FUNCTION_BLOCK _ETcVn2dCodeSearchStrategy_TestSuite EXTENDS TcUnit.FB_TestSuite
VAR
END_VAR

TestAddress();
TestClearReference();
TestClone();
TestTypeNameReturnsExpected();
TestIdentifierReturnsExpected();
TestMakeReferenceToFollowsReference();
TestMakeReferenceToUpdatesReference();
TestSize();
TestValueReturnsExpectedAfterInit();
TestValueReturnsExpectedAfterChange();
TestSerializeTypeWith();
TestSerializeWith();
TestTryDeserializeFrom();
TestTryMakeReferenceToFollowsReference();
TestTryMakeReferenceToUpdatesReference();

METHOD PUBLIC TestAddress
VAR
    _type : _ETcVn2dCodeSearchStrategy(ETcVn2dCodeSearchStrategy.TCVN_CSS_DEFAULT);
    notExpected : PVOID := 0;
    actual : PVOID;
END_VAR
TEST('TestAddress');

actual := _type.Address;

AssertFalse(
    Condition := (notExpected = actual),
    Message := 'Type did not return a valid address.'
);

TEST_FINISHED();
END_METHOD

METHOD PUBLIC TestClearReference
VAR
    _type : _ETcVn2dCodeSearchStrategy(ETcVn2dCodeSearchStrategy.TCVN_CSS_DEFAULT);
	target : ETcVn2dCodeSearchStrategy := ETcVn2dCodeSearchStrategy.TCVN_CSS_DEFAULT;
    expected : ETcVn2dCodeSearchStrategy := ETcVn2dCodeSearchStrategy.TCVN_CSS_DEFAULT;
    actual : ETcVn2dCodeSearchStrategy;
END_VAR
TEST('TestClearReference');

_type.MakeReferenceTo(target);
_type.ClearReference();
target := ETcVn2dCodeSearchStrategy.TCVN_CSS_FIRST_FLIPPED;

actual := _type.Value;

AssertEquals(
    Expected := expected,
    Actual := actual,
    Message := 'Value continued to follow target.'
);

TEST_FINISHED();
END_METHOD

METHOD PUBLIC TestClone
VAR
    _type : _ETcVn2dCodeSearchStrategy(ETcVn2dCodeSearchStrategy.TCVN_CSS_DEFAULT);
	clone : I_Datatype;
	isValidClone : BOOL;
	compareResult : DINT;
END_VAR
TEST('TestClone');

clone := _type.Clone();

isValidClone := clone <> 0;

IF isValidClone THEN
	compareResult := memcmp(_type.Address, clone.Address, clone.Size);
END_IF

AssertTrue(
	Condition := isValidClone,
	Message := 'Clone did not produce a clone'
);

AssertEquals_DINT(
	Expected := 0,
    Actual := compareResult,
    Message := 'Clone did not return a valid clone.'
);

clone.Dispose();

TEST_FINISHED();
END_METHOD

METHOD PUBLIC TestIdentifierReturnsExpected
VAR
    _type : _ETcVn2dCodeSearchStrategy(ETcVn2dCodeSearchStrategy.TCVN_CSS_DEFAULT);
    expected : STRING := 'ETcVn2dCodeSearchStrategy';
    actual : STRING;
END_VAR
TEST('TestIdentifierReturnsExpected');

actual := _type.Identifier;

AssertEquals_STRING(
    Expected := expected,
    Actual := actual,
    Message := 'Type did not return correct iec type.'
);

TEST_FINISHED();
END_METHOD

METHOD PUBLIC TestMakeReferenceToFollowsReference
VAR
    _type : _ETcVn2dCodeSearchStrategy(ETcVn2dCodeSearchStrategy.TCVN_CSS_DEFAULT);
	target : ETcVn2dCodeSearchStrategy := ETcVn2dCodeSearchStrategy.TCVN_CSS_DEFAULT;
    expected : ETcVn2dCodeSearchStrategy := ETcVn2dCodeSearchStrategy.TCVN_CSS_FIRST_FLIPPED;
    actual : ETcVn2dCodeSearchStrategy;
END_VAR
TEST('TestMakeReferenceToFollowsReference');

_type.MakeReferenceTo(target);
target := ETcVn2dCodeSearchStrategy.TCVN_CSS_FIRST_FLIPPED;

actual := _type.Value;

AssertEquals(
    Expected := expected,
    Actual := actual,
    Message := 'Value did not follow target change.'
);

TEST_FINISHED();
END_METHOD

METHOD PUBLIC TestMakeReferenceToUpdatesReference
VAR
    _type : _ETcVn2dCodeSearchStrategy(ETcVn2dCodeSearchStrategy.TCVN_CSS_DEFAULT);
	target : ETcVn2dCodeSearchStrategy := ETcVn2dCodeSearchStrategy.TCVN_CSS_DEFAULT;
    expected : ETcVn2dCodeSearchStrategy := ETcVn2dCodeSearchStrategy.TCVN_CSS_FIRST_FLIPPED;
    actual : ETcVn2dCodeSearchStrategy;
END_VAR
TEST('TestMakeReferenceToUpdatesReference');

_type.MakeReferenceTo(target);
_type.Value := ETcVn2dCodeSearchStrategy.TCVN_CSS_FIRST_FLIPPED;

actual := target;

AssertEquals(
    Expected := expected,
    Actual := actual,
    Message := 'Value did not update target.'
);

TEST_FINISHED();
END_METHOD

METHOD PUBLIC TestSerializeTypeWith
VAR
    _type : _ETcVn2dCodeSearchStrategy(ETcVn2dCodeSearchStrategy.TCVN_CSS_DEFAULT);
    serializer : JsonSerializer;
    expected : STRING(500) := '{"typeName":"ENUM","identifier":"ETcVn2dCodeSearchStrategy","enumerations":["TCVN_CSS_DEFAULT","TCVN_CSS_FIRST_FLIPPED","TCVN_CSS_FIRST_INVERTED","TCVN_CSS_FIRST_NOT_FLIPPED","TCVN_CSS_FIRST_NOT_INVERTED","TCVN_CSS_ONLY_FLIPPED","TCVN_CSS_ONLY_INVERTED","TCVN_CSS_ONLY_NOT_FLIPPED","TCVN_CSS_ONLY_NOT_INVERTED"],"baseType":{"typeName":"UDINT","minValue":0,"maxValue":4294967295,"isSigned":false,"isFloat":false}}';
    actual : STRING(500);
END_VAR
TEST('TestSerializeTypeWith');

serializer.Reset();
_type.SerializeTypeWith(serializer);
serializer.TryGetSerializedData(ADR(actual), SIZEOF(actual));

AssertEquals_STRING(
    Expected := expected,
    Actual := actual,
    Message := 'Serialization of type did not return correct string.'
);

TEST_FINISHED();
END_METHOD

METHOD PUBLIC TestSerializeWith
VAR
    _type : _ETcVn2dCodeSearchStrategy(ETcVn2dCodeSearchStrategy.TCVN_CSS_DEFAULT);
    serializer : JsonSerializer;
    expected : STRING := '"TCVN_CSS_DEFAULT"';
    actual : STRING(500);
END_VAR
TEST('TestSerializeWith');

serializer.Reset();
_type.SerializeWith(serializer);
serializer.TryGetSerializedData(ADR(actual), SIZEOF(actual));

AssertEquals_STRING(
    Expected := expected,
    Actual := actual,
    Message := 'Serialization of type data did not return correct string.'
);

TEST_FINISHED();
END_METHOD

METHOD PUBLIC TestSize
VAR
    _type : _ETcVn2dCodeSearchStrategy(ETcVn2dCodeSearchStrategy.TCVN_CSS_DEFAULT);
    expected : UDINT := SIZEOF(ETcVn2dCodeSearchStrategy);
    actual : UDINT;
END_VAR
TEST('TestSize');

actual := _type.Size;

AssertEquals_UDINT(
    Expected := Expected,
    Actual := actual,
    Message := 'Type did not return the correct size.'
);

TEST_FINISHED();
END_METHOD

METHOD PUBLIC TestTryDeserializeFrom
VAR
    deserializer : JsonDeserializer;
    feedback : DeserializerFeedback;
    json : STRING := '"TCVN_CSS_DEFAULT"';
    _type : _ETcVn2dCodeSearchStrategy(ETcVn2dCodeSearchStrategy.TCVN_CSS_DEFAULT);
    expected : ETcVn2dCodeSearchStrategy := ETcVn2dCodeSearchStrategy.TCVN_CSS_DEFAULT;
    actual : ETcVn2dCodeSearchStrategy;
 END_VAR
TEST('TestTryDeserializeFrom');

deserializer.Reset();
deserializer.TryLoad(json);
_type.TryDeserializeFrom(Deserializer, Feedback);

actual := _type.Value;

AssertEquals(
    Expected := expected,
    Actual := actual,
    Message := 'Type did not deserialize correctly.'
);

TEST_FINISHED();
END_METHOD

METHOD PUBLIC TestTryMakeReferenceToFollowsReference
VAR
    _type : _ETcVn2dCodeSearchStrategy(ETcVn2dCodeSearchStrategy.TCVN_CSS_DEFAULT);
	target : _ETcVn2dCodeSearchStrategy(ETcVn2dCodeSearchStrategy.TCVN_CSS_DEFAULT);
    expected : ETcVn2dCodeSearchStrategy := ETcVn2dCodeSearchStrategy.TCVN_CSS_FIRST_FLIPPED;
    actual : ETcVn2dCodeSearchStrategy;
END_VAR
TEST('TestTryMakeReferenceToFollowsReference');

_type.TryMakeReferenceTo(target);
target.Value := ETcVn2dCodeSearchStrategy.TCVN_CSS_FIRST_FLIPPED;

actual := _type.Value;

AssertEquals(
    Expected := expected,
    Actual := actual,
    Message := 'Value did not follow target change.'
);

TEST_FINISHED();
END_METHOD

METHOD PUBLIC TestTryMakeReferenceToUpdatesReference
VAR
    _type : _ETcVn2dCodeSearchStrategy(ETcVn2dCodeSearchStrategy.TCVN_CSS_DEFAULT);
	target : _ETcVn2dCodeSearchStrategy(ETcVn2dCodeSearchStrategy.TCVN_CSS_DEFAULT);
    expected : ETcVn2dCodeSearchStrategy := ETcVn2dCodeSearchStrategy.TCVN_CSS_FIRST_FLIPPED;
    actual : ETcVn2dCodeSearchStrategy;
END_VAR
TEST('TestTryMakeReferenceToUpdatesReference');

_type.TryMakeReferenceTo(target);
_type.Value := ETcVn2dCodeSearchStrategy.TCVN_CSS_FIRST_FLIPPED;

actual := target.Value;

AssertEquals(
    Expected := expected,
    Actual := actual,
    Message := 'Value did not update target.'
);

TEST_FINISHED();
END_METHOD

METHOD PUBLIC TestTypeNameReturnsExpected
VAR
    _type : _ETcVn2dCodeSearchStrategy(ETcVn2dCodeSearchStrategy.TCVN_CSS_DEFAULT);
    expected : STRING := 'ENUM';
    actual : STRING;
END_VAR
TEST('TestTypeNameReturnsExpected');

actual := _type.TypeName;

AssertEquals_STRING(
    Expected := expected,
    Actual := actual,
    Message := 'Type did not return correct iec type.'
);

TEST_FINISHED();
END_METHOD

METHOD PUBLIC TestValueReturnsExpectedAfterChange
VAR
    _type : _ETcVn2dCodeSearchStrategy(ETcVn2dCodeSearchStrategy.TCVN_CSS_DEFAULT);
    expected : ETcVn2dCodeSearchStrategy := ETcVn2dCodeSearchStrategy.TCVN_CSS_FIRST_FLIPPED;
    actual : ETcVn2dCodeSearchStrategy;
END_VAR
TEST('TestValueReturnsExpectedAfterChange');

_type.Value := ETcVn2dCodeSearchStrategy.TCVN_CSS_FIRST_FLIPPED;

actual := _type.Value;

AssertEquals(
    Expected := expected,
    Actual := actual,
    Message := 'Expected value not returned after change.'
);

TEST_FINISHED();
END_METHOD

METHOD PUBLIC TestValueReturnsExpectedAfterInit
VAR
    _type : _ETcVn2dCodeSearchStrategy(ETcVn2dCodeSearchStrategy.TCVN_CSS_DEFAULT);
    expected : ETcVn2dCodeSearchStrategy := ETcVn2dCodeSearchStrategy.TCVN_CSS_DEFAULT;
    actual : ETcVn2dCodeSearchStrategy;
END_VAR
TEST('TestValueReturnsExpectedAfterInit');

actual := _type.Value;

AssertEquals(
    Expected := expected,
    Actual := actual,
    Message := 'Expected value not returned after Init.'
);

TEST_FINISHED();
END_METHOD

END_FUNCTION_BLOCK

(* stored: Version 1.1.0.1, ProductVersion 3.1.4024.12
   POU _ETcVn2dCodeSearchStrategy_TestSuite: Id {6437228a-7660-4c0d-b535-65226c912a28}, SpecialFunc None
   Method TestAddress: Id {e5d5aed4-c00a-464d-ba41-6f769ea80945}
   Method TestClearReference: Id {ccb49ab5-497b-4333-82a4-81aca560be1f}
   Method TestClone: Id {f7783ad6-e504-428e-81a7-36fba43d27f4}
   Method TestIdentifierReturnsExpected: Id {a1efc315-531e-43d6-867b-93b1ce671e5d}
   Method TestMakeReferenceToFollowsReference: Id {0650108b-4755-438e-927b-085c87025ce2}
   Method TestMakeReferenceToUpdatesReference: Id {cbc88859-d002-4488-a1cd-ab74718af331}
   Method TestSerializeTypeWith: Id {6d5003ca-96e5-4f36-b2d4-4698fbbb9ded}
   Method TestSerializeWith: Id {0424348c-580e-426c-80b3-4549ee87fcf2}
   Method TestSize: Id {61cbb312-d3aa-44da-a97d-d6744bc0f9fb}
   Method TestTryDeserializeFrom: Id {e059d202-2fb1-4651-8a38-34903c6f076a}
   Method TestTryMakeReferenceToFollowsReference: Id {ef1c5f2d-8806-4cc3-8017-8072527a9a84}
   Method TestTryMakeReferenceToUpdatesReference: Id {27fcbde9-ed06-47f1-927e-255f1dcb21a4}
   Method TestTypeNameReturnsExpected: Id {32342309-6455-4ee5-9de0-0de388ad23e9}
   Method TestValueReturnsExpectedAfterChange: Id {5b4a25c8-6319-4a62-9ddd-742820892ed4}
   Method TestValueReturnsExpectedAfterInit: Id {4266e2a4-d664-4809-8133-c205a9712e3b} *)
